(*These are parameters that are used to initiate axis movements
They are commands that are commonly used commands*)
TYPE ST_AxisControl :
STRUCT
    //Actions from controls system
    bExecute: BOOL; //Trigger to execute a motion function block
    bReset: BOOL; //Reset axis from Error state
    bStop: BOOL; //Stop the axis movement
    bHalt: BOOL; //Halt the axis movement
    bEnable: BOOL; //Enable axis drive
    bInterlockFwd: BOOL := FALSE; //Enable interlock for forward movement (resets at end of cycle)
    bInterlockBwd: BOOL := FALSE; //Enable interlock for backward movement (resets at end of cycle)
    eCommand: E_MotionFunctions; //Specifies the motion function to execute
    fVelocity: LREAL; //Specifies the velocity to be used for executing motion commands
    fJogVelocity: LREAL; //Velocity for jogging operations
    fAcceleration: LREAL; //Acceleration for the movement command (0 uses the NC default)
    fDeceleration: LREAL; //Deceleration for the movement command
    fPosition: LREAL; //Target position for absolute moves or distance for relative moves
    bHWMaskActive: BOOL := FALSE; //Indicates if hardware masking is active
    fMaskedTemperature: REAL := 0.0; //Temperature value used when the hardware masking is active
    bPressurizeAirpad AT %Q*: BOOL; //Output from method controlling airpad
    bAirpadManualPressureOn: BOOL := FALSE; //Pressurize airpad manually
    bReleaseBrake AT %Q*: BOOL; //Output from method controlling brake
END_STRUCT
END_TYPE

(* stored: Version 1.1.0.1
   DUT ST_AxisControl: Id {c02b2c99-be98-4acd-b0cb-dc10c1ff77f2} *)
